ABB RobotStudio station: 4230.rsstn

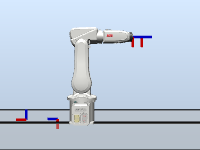
Station Station (saved by RobotStudio 6.7.7936.1011)
Controller MTRN4230
  mechanical unit ROB_1: IRB120_3_58__01, 6 joints, base frame (0, 0, 0) mm
Layout (positions relative to the parent item):
  - IRB120_3_58__01 [mechanism, from Robots\IRB120_3_58_G_01.rslib] at (0, 0, 0) mm; joint values [-1.5708, 0, 0, 0, 0, 0] (rad or m)
Targets, tools, work objects and paths stored in the station, written as RAPID:
! task T_ROB1
MODULE MTRN_Rob_Data
  PERS tooldata tSCup:=[TRUE,[[0,0,65],[1,0,0,0]],[0.5,[0,0,20],[1,0,0,0],0,0,0]];
  PERS wobjdata wTable:=[FALSE,TRUE,"",[[175,0,147],[1,0,0,0]],[[0,0,0],[1,0,0,0]]];
  PERS wobjdata wConv:=[FALSE,TRUE,"",[[50,184,22],[0.5,-0.5,0.5,0.5]],[[1,1,1],[1,0,0,0]]];
  CONST robtarget pTableHome:=[[0,0,0],[1,0,0,0],[0,0,0,0],[9E+09,9E+09,9E+09,9E+09,9E+09,9E+09]];
  CONST jointtarget jtCalibPos:=[[-90,0,0,0,0,0],[9E+09,9E+09,9E+09,9E+09,9E+09,9E+09]];
  PERS wobjdata Workobject_2:=[FALSE,TRUE,"",[[175,0,147],[1,0,0,0]],[[0,0,0],[1,0,0,0]]];
  PERS wobjdata wConveyer:=[FALSE,TRUE,"",[[0,409,22],[0.707106781,0,0,0.707106781]],[[0,0,0],[1,0,0,0]]];
  PERS wobjdata wConveyerCamera:=[FALSE,TRUE,"",[[-71,429,1110],[1,0,0,0]],[[0,0,0],[1,0,0,0]]];
  PERS wobjdata wTableCamera:=[FALSE,TRUE,"",[[309,19,1110],[1,0,0,0]],[[0,0,0],[1,0,0,0]]];
  PERS wobjdata wWorld:=[FALSE,TRUE,"",[[-3025,-3282,-585],[1,0,0,0]],[[0,0,0],[1,0,0,0]]];
  PERS wobjdata wEffector:=[FALSE,TRUE,"",[[401.362715792,45.961925887,184.649812471],[0.277815883,0.115075154,-0.881119559,0.364971733]],[[0,0,0],[1,0,0,0]]];
  PERS wobjdata wBase:=[FALSE,TRUE,"",[[0,0,0],[1,0,0,0]],[[0,0,0],[1,0,0,0]]];
ENDMODULE

! task T_ROB1
MODULE Assignment2
  PERS wobjdata wobjCurrent:=[FALSE,TRUE,"",[[0,0,0],[1,0,0,0]],[[0,0,0],[1,0,0,0]]];
  PROC Main()
    MoveToCalibPos;
    SingArea \Wrist;
    ConfJ \On;
    MoveToPose;
    conRunOn;
    conRunOff;
    conDirHome;
    conDirRob;
    vacSolOn;
    vacSolOff;
    vacPwrOn;
    vacPwrOff;
    MoveToCalibPos;
    vacPwrOff;
    vacSolOff;
    conRunOff;
  ENDPROC
  PROC MoveToPose()
    MoveAbsJ thetas_new_formatted,move_speed,fine,tSCup;
  ENDPROC
  PROC vacPwrOn()
    SetDO DO10_1,1;
  ENDPROC
  PROC vacPwrOff()
    SetDO DO10_1,0;
  ENDPROC
  PROC vacSolOn()
    SetDO DO10_2,1;
  ENDPROC
  PROC vacSolOff()
    SetDO DO10_2,0;
  ENDPROC
  PROC conRunOn()
    SetDO DO10_3,1;
  ENDPROC
  PROC conRunOff()
    SetDO DO10_3,0;
  ENDPROC
  PROC conDirRob()
    SetDO DO10_4,1;
  ENDPROC
  PROC conDirHome()
    SetDO DO10_4,0;
  ENDPROC
ENDMODULE

! task T_ROB1
MODULE MTRN4230_Server_Sample
  PROC MainServer()
    target;
    angles;
    GetIO;
    GetError;
    WaitTime 1;
    CloseConnection;
  ENDPROC
  PROC ListenForAndAcceptConnection()
  ENDPROC
  PROC CloseConnection()
  ENDPROC
  PROC target()
  ENDPROC
  PROC angles()
  ENDPROC
  PROC GetIO()
  ENDPROC
  PROC GetError()
  ENDPROC
ENDMODULE

! task T_ROB1
MODULE MTRN4230_Move_Sample
  PROC MoveJSample()
    MoveJ pTableHome,v100,fine,tSCup;
  ENDPROC
  PROC MoveLSample()
    MoveL Offs(pTableHome, 0, 0, 100),v100,fine,tSCup;
  ENDPROC
  PROC MainMove()
    MoveToCalibPos;
    MoveJSample;
    MoveLSample;
  ENDPROC
ENDMODULE

! task T_ROB1
MODULE MTRN4230_IO_Sample
  PROC MainIO()
    TurnVacOn;
    WaitTime 2;
    TurnVacOff;
    TurnConOnSafely;
    WaitTime 2;
    TurnConOff;
  ENDPROC
  PROC TurnVacOff()
    SetDO DO10_1,0;
  ENDPROC
  PROC TurnConOff()
    SetDO DO10_3,0;
  ENDPROC
  PROC TurnVacOn()
    SetDO DO10_1,1;
  ENDPROC
  PROC TurnConOnSafely()
    SetDO DO10_3,1;
    SetDO DO10_3,0;
  ENDPROC
ENDMODULE

! task T_ROB1
MODULE MTRN_Rob_Proc
  PROC MoveToCalibPos()
    MoveAbsJ jtCalibPos,v400,fine,tool0;
  ENDPROC
ENDMODULE

! task T_ROB1
MODULE <mod2>
  PROC MainAss2()
  ENDPROC
ENDMODULE

